// TIA Portal V18 export
DATA_BLOCK "01_Pushbutton"   // DB2, F_DB
{ S7_Optimized_Access := 'TRUE'; DB_Accessible_From_OPC_UA := 'FALSE' }
VERSION : 0.1
// stored: AutoNumber true, DBAccessibleFromOPCUA false, DBAccessibleFromWebserver true
   VAR
      AlwaysFALSE : Bool;
      AlwaysTRUE : Bool;
      "No Operation" : Bool;
      "Emergency Push Button [ =S1+MS1.CC1-S67001 ]" : Bool;
      "Emergency Push Button [ =S1+PC1.CC1-X80101 ]" : Bool;
      "Emergency Push Button [ =S2+MS2.CC1-S67001 ]" : Bool;
      "Emergency Push Button [ =S2+PC2.CC1-X80101 ]" : Bool;
      "Safety Breaker [ =S1+MS1.CC1-Q67001 ]" : Bool;
      "Safety Breaker [ =S2+MS2.CC1-Q67001 ]" : Bool;
   END_VAR
BEGIN
END_DATA_BLOCK
